{attribute 'qualified_only'}
{attribute 'strict'}
TYPE E_HTTP_CONNECTION :
(
	E_CONNECTION_CLOSE := 0,
	E_CONNECTION_KEEP_ALIVE
);
END_TYPE

(* stored: Version 1.1.0.1, ProductVersion 3.1.4020.3
   DUT E_HTTP_CONNECTION: Id {cc31036e-067c-40e7-8ef0-ebfe7268bd52} *)
